{attribute 'GeneratedUsingTerminal: EL6631-0000-0018'}
{attribute addProperty VendorId "#x00000002"}
{attribute addProperty BoxType "EL6631-0000-0018"}
{attribute addProperty Description "EL6631 PROFINET IO Controller"}
{attribute addProperty Physics "KK"}
{attribute addProperty Id "InfoDataAT %I*InfoData_8F85596B2"}
{attribute addProperty CRC "2699822940"}
{attribute addProperty Size "2"}
TYPE EL6631_A0EC075C EXTENDS TcoIo.EtcSlaveTerminalBase_947E5A46 :
STRUCT
	{attribute addProperty Name "InfoData"}
	InfoData : InfoData_8F85596B;
END_STRUCT
END_TYPE

(* stored: Version 1.2.0.0
   DUT EL6631_A0EC075C: Id {548871ad-9df7-4c64-bda6-008e70ad7a8f} *)
